{attribute 'qualified_only'}
VAR_GLOBAL
	nTest AT %Q* : INT;
END_VAR

(* stored: Version 1.1.0.1, ProductVersion 3.1.4024.12
   GVL Test: Id {c07de636-1422-4c2d-b30a-f7b29aca956d} *)
